// TwinCAT 3 PLC project ePU10V2
// ProgramVersion: 3.1.4026.24
// libraries:
//   Tc2_ControllerToolbox, * (Beckhoff Automation GmbH)
//   Tc2_EtherCAT, * (Beckhoff Automation GmbH)
//   Tc2_ModbusSrv, * (Beckhoff Automation GmbH)
//   Tc2_ProfinetDiag, * (Beckhoff Automation GmbH)
//   Tc2_Standard, * (Beckhoff Automation GmbH)
//   Tc2_SUPS, * (Beckhoff Automation GmbH)
//   Tc2_System, * (Beckhoff Automation GmbH)
//   Tc2_Utilities, * (Beckhoff Automation GmbH)
//   Tc3_EventLogger, * (Beckhoff Automation GmbH)
//   Tc3_IotBase, * (Beckhoff Automation GmbH)
//   Tc3_JsonXml, * (Beckhoff Automation GmbH)
// project tree:
//   DUTs/Enums/ eBatteryType.TcDUT, eForceBool.TcDUT, eGridTripMode.TcDUT, eObject_ID.TcDUT, ePNcouplerType.TcDUT, eSubValues.TcDUT, Phases.TcDUT
//   DUTs/Structs/ ST_AnalogInputData.TcDUT, ST_AnalogInputDiag.TcDUT, ST_Service_DigitalOutIn.TcDUT, ST_Service_DigitalOutInWithDependency.TcDUT, ST_Service_DigitalOutInWithSafety.TcDUT
//   DUTs/System/ ST_System_Config.TcDUT, ST_System_GridcodeParams.TcDUT, ST_System_MachineParams.TcDUT
//   GVLs/ Service.TcGVL, GVL.TcGVL, Settings.TcGVL, Units.TcGVL
//   POUs/Eventlogger/_enum/ eEventLogCategory.TcDUT, eEventLogSeverity.TcDUT
//   POUs/Eventlogger/_structs/ ST_EventLogEntry.TcDUT, ST_EventLogger_Params.TcDUT
//   / PlcTask.TcTTO, MonitorControlTask.TcTTO
//   POUs/ErrorHandling/ ErrorHandling.TcPOU, FB_AddErrorST.TcPOU
//   POUs/ErrorHandling/_enums/ eErrAckAccess.TcDUT, eSeverity.TcDUT
//   POUs/ErrorHandling/_strucs/ ST_ErrorStruct.TcDUT
//   POUs/Functions-FBs-Programs/ fbValueOutOfRange.TcPOU, Fb_BindControlVars.TcPOU, fb_IncrementPowerStep.TcPOU, FB_OverCurrentDetect.TcPOU, fb_Ramp.TcPOU, fb_Ramp_dual.TcPOU, FB_UpperLimitAndTimeExceeded.TcPOU, ITF_StandardFB.TcIO
//   POUs/Functions-FBs-Programs/IO_modules/Beckhoff/ FB_EK1100.TcPOU, FB_EL3453.TcPOU
//   POUs/Functions-FBs-Programs/IO_modules/Beckhoff/Structs/ DataSelector.TcDUT, ST_PQGridQualityData.TcDUT, ST_PQPowerData.TcDUT, ST_PQstatusData.TcDUT, ST_PQVoltageData.TcDUT
//   POUs/Functions-FBs-Programs/_acFunctions/ AcCheck.TcPOU, ACFrequencyCheck.TcPOU, AcPhasesOK.TcPOU, ACVoltageCheck.TcPOU, CurrentToKw.TcPOU, fb_LOMdetection.TcPOU, kWToCurrent.TcPOU, LineUnbalance.TcPOU, PowerFactor.TcPOU, ReactivePower.TcPOU
//   POUs/Functions-FBs-Programs/_generalFunctions/ Between.TcPOU, ConcatMultiString.TcPOU, fb_MovingAverage.TcPOU, FB_StartStop.TcPOU, F_RoundReal.TcPOU, IsNaN.TcPOU, LimitTrigger.TcPOU, Median.TcPOU, PackByte.TcPOU, PackWord.TcPOU, Scale.TcPOU, ValueOutOfRange.TcPOU, WriteOnEdge.TcPOU, XNOR.TcPOU
//   POUs/Functions-FBs-Programs/_PRGS/ SystemClock.TcPOU
//   POUs/ MAIN_Fast.TcPOU, MAIN_Slow.TcPOU
//   POUs/MonitoringControl/ ControlManager.TcPOU, FB_TestScripts.TcPOU
//   POUs/MonitoringControl/ExternalControl/enums/ eExternalControlMode.TcDUT, GenGridMode.TcDUT, uSWversion.TcDUT
//   POUs/MonitoringControl/ExternalControl/ FB_ExtControllerTest.TcPOU, FB_ExternalController.TcPOU
//   POUs/MonitoringControl/ExternalControl/Structs/future use/ ST_PNInput_DCBusExpansion.TcDUT, ST_PNInput_DCCharger.TcDUT, ST_PNInput_ParallelOperation.TcDUT, ST_PNOutput_DCCharger.TcDUT, ST_PNOutput_DCExpansion.TcDUT, ST_PNOutput_ParallelOperation.TcDUT
//   POUs/MonitoringControl/ExternalControl/Structs/NestedStructs/ ST_PNInput_ACDCCharger.TcDUT, ST_PNInput_Battery.TcDUT, ST_PNInput_GenControl.TcDUT, ST_PNInput_General.TcDUT, ST_PNInput_InputField.TcDUT, ST_PNInput_InputGridControl.TcDUT, ST_PNInput_PeakShaveBox.TcDUT, ST_PNInput_Powerstack.TcDUT, ST_PNOutput_ACDCCharger.TcDUT, ST_PNOutput_Battery.TcDUT, ST_PNOutput_GenControl.TcDUT, ST_PNOutput_General.TcDUT, ST_PNOutput_InputField.TcDUT, ST_PNOutput_InputGridControl.TcDUT, ST_PNOutput_OutputField.TcDUT, ST_PNOutput_PeakShaveBox.TcDUT, ST_PNOutput_PowerStack.TcDUT, ST_PNOutput_ZPT.TcDUT
//   POUs/MonitoringControl/ExternalControl/Structs/ ST_Extcontroller_params.TcDUT, ST_PNinput.TcDUT, ST_PNOutput.TcDUT, ST_PNTest.TcDUT
//   POUs/MonitoringControl/HMI/ FB_HMIButtons.TcPOU, HMI.TcPOU
//   POUs/MonitoringControl/HMI/_Structs/ControlStructures/HardSettings %28localOnly%29/ ST_HardSettings.TcDUT (not stored), ST_HardSettings_DCcharger.TcDUT (not stored), ST_HardSettings_ParallelOperation.TcDUT (not stored), ST_HardSettings_PeakshaveBox.TcDUT (not stored), ST_HardSettings_Setup.TcDUT (not stored), ST_HardSettings_System.TcDUT (not stored)
//   POUs/MonitoringControl/HMI/_Structs/ControlStructures/OperationVars/ ST_OperationVars.TcDUT, ST_OperationVars_BMS.TcDUT, ST_OperationVars_DCcharger.TcDUT, ST_OperationVars_Genset.TcDUT, ST_OperationVars_Grid.TcDUT, ST_OperationVars_ParallelOperation.TcDUT, ST_OperationVars_System.TcDUT
//   POUs/MonitoringControl/HMI/_Structs/ControlStructures/SoftSettings %28Local+Extern%29/NestedStructs/ ST_Genset_params.TcDUT (not stored), ST_Genset_setpoints.TcDUT (not stored), ST_Input_breakersettings.TcDUT (not stored), ST_Loadbank_params.TcDUT (not stored), ST_peakshave_setpoints.TcDUT (not stored), ST_ScheduleTimeSlot.TcDUT (not stored)
//   POUs/MonitoringControl/HMI/_Structs/ControlStructures/SoftSettings %28Local+Extern%29/ ST_SoftSettings.TcDUT (not stored), ST_Softsettings_AcDcCharger.TcDUT (not stored), ST_SoftSettings_DcLink.TcDUT (not stored), ST_SoftSettings_Genset.TcDUT (not stored), ST_SoftSettings_Grid.TcDUT (not stored), ST_SoftSettings_PeakshaveBox.TcDUT (not stored), ST_SoftSettings_Setup.TcDUT (not stored), ST_SoftSettings_System.TcDUT (not stored)
//   POUs/MonitoringControl/HMI/_Structs/ControlStructures/ ST_ControlsHMIonly.TcDUT, ST_ControlVars.TcDUT
//   POUs/MonitoringControl/HMI/_Structs/MonitoringStructures/ ST_HMIdata.TcDUT, ST_HMI_ConditionalFormatting.TcDUT, ST_HMI_Monitor_AcDcCharger.TcDUT, ST_HMI_Monitor_Arraydata.TcDUT, ST_HMI_Monitor_ArrayDataFormat.TcDUT, ST_HMI_Monitor_Battery.TcDUT, ST_HMI_Monitor_Connections.TcDUT, ST_HMI_Monitor_CoolingSystem.TcDUT, ST_HMI_Monitor_DcLink.TcDUT, ST_HMI_Monitor_Enclosure.TcDUT, ST_HMI_Monitor_FireDetection.TcDUT, ST_HMI_Monitor_IPSU.TcDUT, ST_HMI_Monitor_Limits.TcDUT, ST_HMI_Monitor_OCP.TcDUT, ST_HMI_Monitor_Powerstack.TcDUT, ST_HMI_Monitor_Protections.TcDUT, ST_HMI_Monitor_PSB.TcDUT, ST_HMI_Monitor_switchgear.TcDUT, ST_HMI_Monitor_System.TcDUT, ST_HMI_Monitor_UPS.TcDUT, ST_HMI_Monitor_ZPT.TcDUT, ST_HMI_PowerMeas.TcDUT, ST_HMI_PowerMeasDC.TcDUT
//   POUs/MonitoringControl/HMI/_Structs/ ST_HMI_Control.TcDUT, ST_HMI_Historize.TcDUT, ST_HMI_Monitor.TcDUT
//   POUs/MonitoringControl/IoT/DUTS/ eConnectionState.TcDUT, eDataMappingVarNames.TcDUT, eIoTCommVersion.TcDUT, eLogType.TcDUT, eUpdate.TcDUT, e_ORAttributeType.TcDUT, ST_AutoProvisioning.TcDUT, ST_IotProps.TcDUT, ST_RW.TcDUT, ST_Supervisor.TcDUT, ST_VarBuffer.TcDUT
//   POUs/MonitoringControl/IoT/ FB_IotController.TcPOU, MqttComOpenremote.TcPOU, RestComOpenremote.TcPOU
//   POUs/MonitoringControl/IoT/_Structs/ ST_IoTDataHMI.TcDUT, ST_IotData_credits.TcDUT, st_IOT_params.TcDUT, ST_IOT_SentStateLog.TcDUT
//   POUs/MonitoringControl/_Enums/ eAcInputType.TcDUT, eCapTestSTate.TcDUT, eControlSources.TcDUT, eDcInputType.TcDUT, eEarthingSystems.TcDUT, eGridFormingMode.TcDUT, eGridMode.TcDUT, eNetContactorDirection.TcDUT, eOperationMode.TcDUT, ePeakshaveMode.TcDUT, ePowerControlType.TcDUT, eSchedulerMode.TcDUT, eSystemState.TcDUT, eUgridPowerMode.TcDUT
//   POUs/MonitoringControl/_Structs/ ST_ExtController_Events.TcDUT, ST_ExtController_get.TcDUT, ST_ExtController_limits.TcDUT, ST_ExtController_Set.TcDUT, ST_PLCPersistentVars.TcDUT
//   POUs/Objects/4Grouter/Struct/ ST_router_service.TcDUT, dwtoreal.TcDUT, eModemState.TcDUT, eNetworkState.TcDUT, eSimSelectionMode.TcDUT, eSimState.TcDUT, eSMSStatus.TcDUT, eWifiSecurityTypes.TcDUT, eWifiStatus.TcDUT, st_Device.TcDUT, st_GPS.TcDUT, st_mobile.TcDUT, st_Router_Events.TcDUT, st_router_get.TcDUT, ST_Router_params.TcDUT, ST_Router_set.TcDUT, st_Wifi.TcDUT
//   POUs/Objects/ACDCCharger/Structs/ ST_ACDCCharger_Service.TcDUT, ST_ACDCCharger_events.TcDUT, ST_ACDCCharger_get.TcDUT, ST_ACDCCharger_params.TcDUT, ST_ACDCCharger_set.TcDUT, ST_SystemDiagnostic.TcDUT, ST_SystemEval.TcDUT
//   POUs/Objects/BMS/eNums/ eBMS_Status.TcDUT, eHVDC_Powerstatus.TcDUT, ePOUState.TcDUT, ePowerControl.TcDUT, ePowerOnStatus.TcDUT
//   POUs/Objects/BMS/ FB_BMS.TcPOU, FB_BMS_IO.TcPOU
//   POUs/Objects/BMS/Structs/ st_BMS_BatterySummary.TcDUT, st_BMS_Events.TcDUT, st_BMS_Get.TcDUT, st_BMS_Params.TcDUT, ST_BMS_Service.TcDUT, st_BMS_Set.TcDUT, st_MBMU_BatterySummary.TcDUT, st_MBMU_Status.TcDUT, st_SBMU_BatterySummary.TcDUT, st_SBMU_Status.TcDUT
//   POUs/Objects/CoolingSystem/enums/ eConditioningRequirement.TcDUT, eCoolingSystemState.TcDUT, eHeatPumpMode.TcDUT, eHeatPumpState.TcDUT, eSupportedHeatpumps.TcDUT
//   POUs/Objects/CoolingSystem/ FB_CoolingSystem.TcPOU, FB_LGThermaV.TcPOU, ITF_Heatpump.TcIO
//   POUs/Objects/CoolingSystem/structs/ LG_Coils.TcDUT, LG_ControlRegs.TcDUT, LG_InputRegs.TcDUT, LG_Statusbits.TcDUT, ST_CoolingSystem_Events.TcDUT, ST_CoolingSystem_Get.TcDUT, ST_CoolingSystem_MaintenanceParams.TcDUT, ST_Coolingsystem_params.TcDUT, ST_HeatpumpData.TcDUT, ST_HeatPumpEvents.TcDUT, ST_HeatPump_Get.TcDUT, st_TCME31_get_1.TcDUT, st_TCME31_Set_1.TcDUT
//   POUs/Objects/DCLink/ FB_CNV520.TcPOU, FB_DCLink.TcPOU, FB_ShuntBournsSSD.TcPOU
//   POUs/Objects/DCLink/_Enums/ eDcLinkState.TcDUT, eDCpowerPriority.TcDUT
//   POUs/Objects/DCLink/_Structs/ ST_Bourns_errors.TcDUT, ST_Bourns_Powerdata.TcDUT, ST_DCLink_events.TcDUT, ST_DCLink_Get.TcDUT, ST_DCLink_IO.TcDUT, ST_DCLink_params.TcDUT, ST_DCLink_set.TcDUT, st_Pixsys.TcDUT
//   POUs/Objects/PowerQualityMonitor/ FB_EastronSDM630.TcPOU, FB_PowerQualityMonitoring.TcPOU
//   POUs/Objects/PowerQualityMonitor/_Enums/ eACRotationState.TcDUT
//   POUs/Objects/PowerQualityMonitor/_Structs/ ST_PowerMonitor_BESS.TcDUT, ST_PowerMonitor_Events.TcDUT, ST_PowerMonitor_get.TcDUT, ST_PowerMonitor_InputField.TcDUT, ST_PowerMonitor_OutputField.TcDUT
//   POUs/Objects/PowerStack/NetContactor/_Structs/ ST_Netcontactor_service.TcDUT, ST_Netcontactor_Events.TcDUT, ST_Netcontactor_get.TcDUT, ST_Netcontactor_set.TcDUT
//   POUs/Objects/PowerStack/_Structs/ ST_Powermodule_Service.TcDUT, ST_Powerstack_MaintenanceParams.TcDUT, ST_Powerstack_Service.TcDUT, ST_PowerModule_calibration.TcDUT, ST_PowerModule_get.TcDUT, ST_PowerModule_params.TcDUT, ST_PowerModule_set.TcDUT, ST_Powerstack_Calibration.TcDUT, ST_PowerStack_get.TcDUT, ST_Powerstack_LOMParams.TcDUT, ST_PowerStack_params.TcDUT, ST_PowerStack_Set.TcDUT
//   POUs/Safety/ Safety.TcPOU, ST_Safety_ContactorEDM.TcDUT, ST_Safety_get.TcDUT, ST_Safety_ToSafetyPrg.TcDUT
//   POUs/Objects/4Grouter/ FB_Teltonika.TcPOU
//   POUs/Objects/ACDCCharger/Enums/ eAcDcChargerState.TcDUT
//   POUs/Objects/ACDCCharger/ FB_AcDcCharger.TcPOU
//   POUs/Objects/ACDCCharger/Structs/Hadi/ E_ChargerState.TcDUT, ST_CanId.TcDUT, ST_ChargerControl.TcDUT, ST_Control.TcDUT, ST_Data.TcDUT, ST_ModuleControl.TcDUT, ST_ModuleData.TcDUT, ST_ModuleStatus.TcDUT
//   POUs/Objects/ACSwitchgear %28clientbox%29/ FB_ACSwitchgear.TcPOU (not stored), ST_ACswitchgear_events.TcDUT (not stored), ST_ACSwitchgear_Get.TcDUT (not stored), ST_ACswitchgear_IO.TcDUT (not stored), ST_ACswitchgear_params.TcDUT (not stored), ST_ACswitchgear_set.TcDUT (not stored)
//   POUs/Objects/Enclosure/Climate/ FB_EnclosureClimate.TcPOU, ST_Enclosureclimate_events.TcDUT, ST_EnclosureClimate_get.TcDUT, ST_EnclosureClimate_Params.TcDUT
//   POUs/Objects/Enclosure/Doors/ FB_DoorsNLocks.TcPOU, ST_DoorsNLocks_get.TcDUT
//   POUs/Objects/Enclosure/ FB_Enclosure.TcPOU
//   POUs/Objects/Enclosure/LedIndicator/BeckhoffController/ eDCstate.TcDUT, eLEDSteps.TcDUT, eSystemStatus.TcDUT, FB_LedBeckhoff.TcPOU, LEDColor.TcDUT, LEDCommands.TcDUT, LEDControl.TcDUT, LEDStatus.TcDUT
//   POUs/Objects/Enclosure/LedIndicator/ eColorOrder.TcDUT, FB_Ledstrip.TcPOU, ST_Ledstrip_get.TcDUT, st_Ledstrip_MachineData.TcDUT, st_Ledstrip_params.TcDUT
//   POUs/Objects/Enclosure/_struct/ ST_Enclosure_get.TcDUT, st_Enclosure_params.TcDUT, ST_enclosure_set.TcDUT
//   POUs/Objects/GenComm/eNums/ eGenControlProtocol.TcDUT, eGenOperationMode.TcDUT, eOnOffState.TcDUT
//   POUs/Objects/GenComm/ FB_AGC150.TcPOU, FB_GenComm.TcPOU
//   POUs/Objects/GenComm/Structs/ ST_AGC150_Set.TcDUT, ST_GenComm_Params.TcDUT, ST_Genset_Get.TcDUT, ST_Genset_Set.TcDUT
//   POUs/Objects/HartingIO/ FB_HartingIO.TcPOU, ST_HartingIO_get.TcDUT, ST_HartingIO_params.TcDUT, ST_HartingIO_set.TcDUT
//   POUs/Objects/HartingIO/_Enum/ eAOTarget.TcDUT, eInputSignal.TcDUT, eOutputContactSignal.TcDUT
//   POUs/Objects/InterMachineCom/ FB_ConnectMqttBroker.TcPOU, FB_InterMachineCommunication.TcPOU, ST_InterMachineCom_Master.TcDUT, ST_IntermachineCom_params.TcDUT, st_InterMachineCom_Slave.TcDUT, ST_InterMachineCom_SlaveConData.TcDUT
//   POUs/Objects/InternalPowerSupply/eNums/ e400VSupplySource.TcDUT, eSupplyState.TcDUT
//   POUs/Objects/InternalPowerSupply/ FB_InternalPowerSupply.TcPOU, FB_InternalPowerSupply_IO.TcPOU
//   POUs/Objects/InternalPowerSupply/Structs/ ST_InternalPowerStatus.TcDUT, ST_InternalPowerSupply_Events.TcDUT, ST_InternalPowerSupply_Get.TcDUT, ST_InternalPowerSupply_Params.TcDUT, ST_InternalPowerSupply_PowerDemand.TcDUT
//   POUs/Objects/InternalPowerSupply/UPS/eNums/ eUPSState.TcDUT
//   POUs/Objects/InternalPowerSupply/UPS/ FB_UPS.TcPOU
//   POUs/Objects/InternalPowerSupply/UPS/Structs/ ST_UPSData.TcDUT, ST_UPSEvents.TcDUT, ST_UPSGET.TcDUT
//   POUs/Objects/NeutralTransformer/ FB_NeutralTransformer.TcPOU, FB_NeutralTransformer_IO.TcPOU
//   POUs/Objects/NeutralTransformer/_Struct/ ST_NeutralTransformer_events.TcDUT, ST_NeutralTransformer_Get.TcDUT, ST_Neutraltransformer_params.TcDUT
//   POUs/Objects/PeakshaveBox/DUTs/ ePSBMode.TcDUT
//   POUs/Objects/PeakshaveBox/ FB_PeakshaveBox.TcPOU, ST_PeakShaveBox_Get.TcDUT, ST_peakshavebox_params.TcDUT, ST_PeakshaveBox_Set.TcDUT
//   POUs/Objects/PLCStatus/Enum/ eFTPState.TcDUT, eInstalState.TcDUT, eNetcomState.TcDUT
//   POUs/Objects/PLCStatus/ FB_PLCState.TcPOU, FB_PLCUpdate.TcPOU, ST_EL9410.TcDUT, ST_PLCstate_get.TcDUT, ST_PLC_events.TcDUT
//   POUs/Objects/PowerStack/ FB_PowerStack.TcPOU
//   POUs/Objects/PowerStack/NetContactor/ eNetcontMode.TcDUT, FB_NetContactor.TcPOU, FB_NetContactor_IO.TcPOU
//   POUs/Objects/PowerStack/PowerModule/ FB_PowerModule.TcPOU, FB_Powermodule_additionalMeasurements.TcPOU, FB_PowerModule_Buscoupler.TcPOU, FB_PowerModule_Inverter.TcPOU
//   POUs/Objects/PowerStack/_Enums/ eInverterModes.TcDUT, eNetContactorState.TcDUT, ePLM.TcDUT, ePowerModes.TcDUT, ePowerModuleThrottlingState.TcDUT, ePowerstate.TcDUT, eStatusPowerModule.TcDUT, eStatusPowerStack.TcDUT
//   POUs/Objects/PowerStack/_Structs/NestedStructs/ ST_InverterControlWord.TcDUT, ST_Inverter_additionalTemperatures.TcDUT, ST_Inverter_LineState.TcDUT, ST_Inverter_StatusWord.TcDUT, ST_Inverter_UgridStatusWord.TcDUT, ST_Inverter_Write.TcDUT, ST_Powermodule_CalibData.TcDUT, ST_Powermodule_Events.TcDUT, ST_Powermodule_PowerCurveCoefficients.TcDUT, ST_PowerStack_Events.TcDUT, ST_Powerstack_ShiftingParams.TcDUT
//   POUs/Objects/ProtectionSystems/ FB_ProtectionSystems.TcPOU
//   POUs/Objects/ProtectionSystems/FireDetection/ FB_FireDetection.TcPOU, FB_FireDetection_IO.TcPOU
//   POUs/Objects/ProtectionSystems/FireDetection/_Enums/ eCOAlarmStatus.TcDUT, eSmokeDetectAlarmStatus.TcDUT
//   POUs/Objects/ProtectionSystems/FireDetection/_Structs/ ST_CODetectors.TcDUT, ST_FireDetection_get.TcDUT, st_Firedetection_params.TcDUT, ST_FireDetection_set.TcDUT, ST_FireSystem_Events.TcDUT, ST_SmokeDetectors.TcDUT, ST_SmokeDetIO.TcDUT
//   POUs/Objects/ProtectionSystems/InsulationMonitoring/ FB_InsulationMonitor.TcPOU
//   POUs/Objects/ProtectionSystems/InsulationMonitoring/_Structs/ ST_InsulationMonitor_get.TcDUT, ST_InsulationMonitor_params.TcDUT, St_InsulationMonitor_PassThrough.TcDUT, ST_InsulationMonitor_set.TcDUT
//   POUs/Objects/ProtectionSystems/OvercurrentProtection/ FB_OvercurrentProtection.TcPOU
//   POUs/Objects/ProtectionSystems/OvercurrentProtection/_Structs/ ST_OvercurrentProtection_Events.TcDUT, ST_OvercurrentProtection_get.TcDUT, ST_OvercurrentProtection_InternalLinking.TcDUT, ST_OvercurrentProtection_Params.TcDUT, ST_OvercurrentProtection_set.TcDUT
//   POUs/Objects/ProtectionSystems/ResidualCurrentMonitoring/ FB_RCMonitor.TcPOU
//   POUs/Objects/ProtectionSystems/ResidualCurrentMonitoring/_Structs/ ST_ResidualCurrentMonitor_get.TcDUT
//   POUs/Objects/ProtectionSystems/SurgeProtection/ FB_SurgeProtection.TcPOU
//   POUs/Objects/ProtectionSystems/SurgeProtection/_Structs/ ST_Surgeprotection_get.TcDUT
//   POUs/Objects/ProtectionSystems/_Struct/ ST_ProtectionSystems_get.TcDUT, ST_ProtectionSystems_Params.TcDUT, ST_ProtectionSystems_set.TcDUT
//   POUs/Objects/RemoteIO/ FB_TruCompTCME21_IOModule.TcPOU, st_TCME31_get.TcDUT, st_TCME31_Set.TcDUT
//   POUs/Objects/WearLogging/ eEntryType.TcDUT, eLogItemGroupID.TcDUT, eLogTypes.TcDUT, FB_Varlogger.TcPOU, LogState.TcDUT, WearLogging.TcPOU
//   POUs/System/ FB_SystemControl.TcPOU
//   POUs/Eventlogger/ FB_Eventlogger.TcPOU, FB_EventLogClient.TcPOU
//   POUs/System/GenGridControl/ FB_ContactorControl.TcPOU, FB_GenGridController.TcPOU
//   POUs/System/GenGridControl/_enums/ eBreakerOperationMode.TcDUT, eGenGridState.TcDUT, eGenIsoInverterMode.TcDUT, eGensetMode.TcDUT, eGensetStartStop.TcDUT, ePowerControlMode.TcDUT, eRunCondition.TcDUT
//   POUs/System/GenGridControl/_structs/ ST_ContactorControl_params.TcDUT, ST_GenGridController_Events.TcDUT, ST_GenGridController_get.TcDUT, ST_GenGridController_Params.TcDUT, St_GenGridController_ParamsGenset.TcDUT, ST_GenGridController_SyncData.TcDUT
//   POUs/System/PowerControl/ fb_measurementCheck.TcPOU, FB_PowerControl.TcPOU
//   POUs/System/PowerControl/_enums/ ePIDmode.TcDUT
//   POUs/System/PowerControl/_Structs/ ST_PowerControl_Events.TcDUT, ST_PowerControl_Get.TcDUT, st_Powercontrol_params.TcDUT, st_Powercontrol_PIDparams.TcDUT, ST_PowerControl_PsTarget_Measurements.TcDUT, ST_Powercontrol_set.TcDUT, ST_PowerControl_SocDroopParams.TcDUT, ST_PowerControl_Target.TcDUT
//   POUs/System/_Structs/ ST_SystemTime.TcDUT, ST_System_Calibration.TcDUT, ST_System_Control.TcDUT, ST_System_Events.TcDUT, ST_System_get.TcDUT, ST_System_Monitor.TcDUT, ST_System_params.TcDUT, ST_System_Properties.TcDUT, ST_System_set.TcDUT
// real-time tasks:
//   TASK FastTask: cycle T#1ms, priority 4, ADS port 350
//   TASK SlowTask: cycle T#10ms, priority 8, ADS port 351
// I/O:
//   DEVICE InternalBus (EtherCAT), AmsNetId 10.46.35.98.2.1
//     Main PLC [EK1200-5000 EtherCAT Power supply (2A E-Bus)]
//       Term 34 (EL6070-0033) [EL6070-0033 1Ch. Licence key terminal, individual licences]
//       Term 2 (EL1809) [EL1809 16Ch. Dig. Input 24V, 3ms]
//       Term 3 (EL2809) [EL2809 16Ch. Dig. Output 24V, 0.5A]
//       Term 4 (EL2809) [EL2809 16Ch. Dig. Output 24V, 0.5A]
//       Term 38 (EL3124-0090) [EL3124-0090 4Ch. Ana. Input 4-20mA, Diff., TwinSAFE SC]
//         modules: Module 1 (TwinSAFE Single Channel)
//       Term 6 (EL3214) [EL3214 4Ch. Ana. Input PT100 (RTD)]
//       Term 7 (EL2574) [EL2574 4 Ch. Pixel LED Controller] (disabled)
//         modules: SlotGroup 1 (Slot 1, 2), SlotGroup 1 (Slot 1, 2), SlotGroup 1 (Slot 1, 2), SlotGroup 1 (Slot 1, 2), SlotGroup 2 (Slot 3, 4), SlotGroup 2 (Slot 3, 4), SlotGroup 2 (Slot 3, 4), SlotGroup 2 (Slot 3, 4)
//       Term 9 (EL1918) [EL1918, 8Ch. Safety Input 24V, TwinSAFE]
//         modules: Module 2 (FSLOGIC)
//       Term 10 (EL2904) [EL2904, 4 Ch. Safety Output 24V, 0.5A, TwinSAFE]
//         modules: Module 1 (FSOES), Module 2 (DO)
//       Term 11 (EK1122) [EK1122 2 port EtherCAT junction]
//       Term 12 (EL9011) [EL9011 End Terminal]
//     Clientpanel-input-IO [EK1101 EtherCAT Coupler (2A E-Bus, ID switch)]
//       Term 26 (EL3453-0020) [EL3453 3Ch. Power Measuring calibrated]
//       Term 27 (EL9011) [EL9011 End Terminal]
//     Doorswitch-IO [EK1101 EtherCAT Coupler (2A E-Bus, ID switch)]
//       Term 24 (EL1008) [EL1008 8Ch. Dig. Input 24V, 3ms]
//       Term 25 (EL9011) [EL9011 End Terminal]
//     Clientpanel-output-IO [EK1101 EtherCAT Coupler (2A E-Bus, ID switch)]
//       Term 13 (EL3453-0020) [EL3453 3Ch. Power Measuring calibrated]
//       Term 21 (EL1809) [EL1809 16Ch. Dig. Input 24V, 3ms]
//       Term 22 (EL2809) [EL2809 16Ch. Dig. Output 24V, 0.5A]
//       Term 23 (EL9011) [EL9011 End Terminal]
//     ACDCcharger-IO [EK1101 EtherCAT Coupler (2A E-Bus, ID switch)]
//       Term 28 (EL6751) [EL6751 CANopen Master]
//       Term 29 (EL9011) [EL9011 End Terminal]
//   DEVICE Device 2 (Profinet Controller), AmsNetId 10.46.35.98.3.1
//     quint4-ups [Phoenix Contact PROFINET IO - Uninterruptible Power Supply 2907079]
//       modules: Term 5 (DAP Module), Term 6 (QUINT4-UPS 24DC/40)
//     pm1buscoupler [Beckhoff Automation PROFINET I/O - EtherCAT coupler, IRT, V2.43, port diagnostic, shared device and system redundancy supported EK9320]
//       modules: Term 1 (DAP Module), Term 3 (EL1008), Term 2 (EL2008), Term 8 (EL3208), Term 8 (EL3208)_1, Term 8 (EL3208)_2, Term 8 (EL3208)_3, Term 8 (EL3208)_4
//     arfif106-1 [VACON VACON OPTE9 Dual-port Ethernet OPTE9]
//       modules: Term 7 (DAP Module), Term 4 (Vendor 4 + 16 PD)
//   DEVICE Device 3 (EL6751), AmsNetId 10.46.35.98.4.1
//     Box 1 (CAN Interface)
//   DEVICE ExternalBus (EtherCAT), AmsNetId 10.46.35.98.5.1
//     PSB_V1 [EK1101 EtherCAT Coupler (2A E-Bus, ID switch)]
//       Term 31 (EL3453) [EL3453 3Ch. Power Measuring]
//       Term 32 (EL9011) [EL9011 End Terminal]
// variable links:
//   InternalBus (EtherCAT) <-> InternalBus (EtherCAT)/Main PLC/Term 10 (EL2904)
//     Main PLC/Term 9 (EL1918)/ConnectionInputs/TwinSafeGroup1.Term 10 (EL2904) - Module 1 (FSOES)_13 TxPDO <-> Module 1 (FSOES)/RxPDO/FSOE
//     Main PLC/Term 9 (EL1918)/ConnectionOutputs/TwinSafeGroup1.Term 10 (EL2904) - Module 1 (FSOES)_13 RxPDO <-> Module 1 (FSOES)/TxPDO/FSOE
//   InternalBus (EtherCAT) <-> InternalBus (EtherCAT)/Main PLC/Term 9 (EL1918)
//     Main PLC/Term 38 (EL3124-0090)/Module 1 (TwinSAFE Single Channel)/TSC Inputs/TSC <-> ConnectionOutputs/TwinSafeGroup1.Term 38 (EL3124-0090) - Module 1 (TwinSAFE Single Channel)_15 RxPDO
//     Main PLC/Term 38 (EL3124-0090)/Module 1 (TwinSAFE Single Channel)/TSC Outputs/TSC <-> ConnectionInputs/TwinSafeGroup1.Term 38 (EL3124-0090) - Module 1 (TwinSAFE Single Channel)_15 TxPDO

CONFIGURATION ePU10V2
    RESOURCE PLC ON TwinCAT3
        TASK PlcTask(INTERVAL := T#1ms, PRIORITY := 4);
        TASK MonitorControlTask(INTERVAL := T#10ms, PRIORITY := 8);
        PROGRAM MAIN_Fast WITH PlcTask : MAIN_Fast;
        PROGRAM MAIN_Slow WITH MonitorControlTask : MAIN_Slow;
    END_RESOURCE
END_CONFIGURATION

// ---- DUTs/Enums/eBatteryType.TcDUT
{attribute 'qualified_only'}
{attribute 'strict'}
TYPE eBatteryType :
(
	standard_306Ah := 0,
	highpower_280Ah := 1
);
END_TYPE

// ---- DUTs/Enums/eForceBool.TcDUT
{attribute 'qualified_only'}
{attribute 'strict'}
{attribute 'to_string'}
TYPE eForceBool:
(
	none := 0,
	On	:= 1,
	Off := 2
);
END_TYPE

// ---- DUTs/Enums/eGridTripMode.TcDUT
{attribute 'qualified_only'}
{attribute 'strict'}
TYPE eGridTripMode :
(
	Gridcode := 500,
	Default	:= 30,
	UPS		:= 10	
) UINT; //milliseconds
END_TYPE

// ---- DUTs/Enums/eObject_ID.TcDUT
{attribute 'qualified_only'}
{attribute 'to_string'}
TYPE eObject_ID :
(	
	None					:= 0,
	Safety					:= 10,
	PowerStack				:= 100,
	NetContactor			:= 150,
	PowerModuleMaster 		:= 200,
	PowerModuleSlave 		:= 300,
	PowerMonitor			:= 400,
	InternalPowerSupply		:= 500,
	UPS						:= 550,
	NeutralTransformer		:= 600,
	HartingIO				:= 650,
	Battery					:= 700,
	Cooling					:= 800,
	HeatPump				:= 850,
	AC_Switchgear			:= 900,
	DC_Switchgear			:= 950,
	RCM						:= 1000,
	SurgeProtection			:= 1010,
	InsulationMonitor		:= 1020,
	Firedetection			:= 1030,
	OCP						:= 1050,
	Enclosure_LED			:= 1200,
	Enclosure_doors			:= 1210,
	Enclosure_climate		:= 1220,
	PLC						:= 2000,
	Router					:= 2100,
	PNcontroller			:= 2200,
	IotController			:= 2300,
	PeakshaveBox			:= 2400,
	ACDCCharger				:= 2500,
	RemoteIO				:= 2600,
	GenGridController		:= 3000,
	PowerController			:= 3100,
	System					:= 3200,
	Genset					:= 4000
	
) WORD := None;
END_TYPE

// ---- DUTs/Enums/ePNcouplerType.TcDUT
{attribute 'qualified_only'}
{attribute 'strict'}

TYPE ePNcouplerType :
(
	None := 0,
	ModbusTCP:= 1,
	Profinet := 2,
	ModbusTCPV2 := 3
);
END_TYPE

// ---- DUTs/Enums/eSubValues.TcDUT
{attribute 'qualified_only'}
{attribute 'strict'}
TYPE eSubValues :
(
	Minimum := 0,
	Average := 1,
	Maximum := 2
);
END_TYPE

// ---- DUTs/Enums/Phases.TcDUT
{attribute 'qualified_only'}
{attribute 'strict'}
{attribute 'to_string'}
TYPE Phases :
(
	AVG 		:= 0,
	L1 			:= 1,
	L2 			:= 2,
	L3 			:= 3,
	N 			:= 4,
	minimum		:= 5,
	maximum		:= 6,
	Sum			:= 7
) INT;
END_TYPE

// ---- DUTs/Structs/ST_AnalogInputData.TcDUT
TYPE ST_AnalogInputData :
STRUCT
	Value			: INT;
	Status			: ST_AnalogInputDiag;
END_STRUCT
END_TYPE

// ---- DUTs/Structs/ST_AnalogInputDiag.TcDUT
TYPE ST_AnalogInputDiag :
STRUCT
	Underrange			: BIT;
	Overrange			: BIT;
	Error				: BIT;
END_STRUCT 
END_TYPE

// ---- DUTs/Structs/ST_Service_DigitalOutIn.TcDUT
TYPE ST_Service_DigitalOutIn :
STRUCT
	Force				: eForceBool; //write value
	Feedback			: BOOL; // readvalue
END_STRUCT
END_TYPE

// ---- DUTs/Structs/ST_Service_DigitalOutInWithDependency.TcDUT
TYPE ST_Service_DigitalOutInWithDependency EXTENDS ST_Service_DigitalOutIn:
STRUCT
	{attribute 'TcHmiSystemEng.Parameter.Name' := 'Dependency state'}
	DependencyOK			: BOOL; 
END_STRUCT
END_TYPE

// ---- DUTs/Structs/ST_Service_DigitalOutInWithSafety.TcDUT
TYPE ST_Service_DigitalOutInWithSafety EXTENDS ST_Service_DigitalOutIn:
STRUCT
	{attribute 'TcHmiSystemEng.Parameter.Name' := 'Dependency state'}
	SafetyLoopOK			: BOOL; 
	EDM					: BOOL;
END_STRUCT
END_TYPE

// ---- DUTs/System/ST_System_Config.TcDUT
TYPE ST_System_Config :
STRUCT
	DefaultSettingsActive			: BOOL := TRUE; //To verify when all settings have been reset.
	b_DoublePowerModule				: BOOL := FALSE;
	b_PeakshaverBoxEnable			: BOOL := FALSE;
	
	//NeutralTransformer
	b_NeutralTransformer			: BOOL := FALSE;
	
	
	//Netcontactor
	b_AutomaticACrotation			: BOOL := FALSE;
	
	//DC
	b_DCbuscoupling					: BOOL := FALSE;
	b_DcCharger						: BOOL := FALSE;
	
	//AC
	b_ACInputConnection				: BOOL := FALSE;
	b_ThirdOutputConnection			: BOOL := FALSE;
	//communication
	e_PNcouplerType					: ePNcouplerType := ePNcouplerType.None;
	
	//batteries
	by_NoBatteryStrings			 	: BYTE := 3; // pieces
	e_BatteryType					: eBatteryType := eBatteryType.standard_306Ah;
	
	//Powernet option
	b_PowernetClient				: BOOL :=  FALSE;
	
	//CLIENT specifics
	b_ClientHMI						: BOOL := FALSE;
	
END_STRUCT
END_TYPE

// ---- DUTs/System/ST_System_GridcodeParams.TcDUT
TYPE ST_System_GridcodeParams :
STRUCT
	r_GridNominalVoltage				: REAL := 400; //VAC
	r_GridNominalFrequency				: REAL := 50; // Hz
	r_GridVoltageMin					: REAL := 360;
	r_GridvoltageMax					: REAL := 440;
	r_GridFrequencyMin					: REAL := 48.5;
	r_GridFrequencyMax					: REAL := 51.5;
	r_CurrentUnbalanceLimit				: REAL := 50;  //%
	ui_GCokReleaseTime					: UINT := 60; //seconds
	ui_GCTripMaxTripTime				: UINT := 40; // milliseconds
END_STRUCT
END_TYPE

// ---- DUTs/System/ST_System_MachineParams.TcDUT
TYPE ST_System_MachineParams :
STRUCT
	BMS									: ST_BMS_params;
	ACDCCharger							: ST_ACDCCharger_params;
	Interpowersupply					: ST_InternalPowerSupply_Params;
	Powerstack							: ST_Powerstack_Params;
	Coolingsystem						: ST_Coolingsystem_Params;
	NeutralTransformer					: ST_Neutraltransformer_Params;
	Protections							: ST_Protectionsystems_Params;
	Enclosure							: ST_Enclosure_Params;
	system								: ST_System_params;
	IOT									: ST_IOT_params;
	Router								: ST_Router_params;
	PSB									: ST_peakshavebox_params;
	ACswitchgear						: ST_ACswitchgear_params;
	HartingIO							: ST_HartingIO_params;
	GenComm								: ST_GenComm_params;
	Eventlogger							: ST_EventLogger_params;
	DC									: ST_DClink_params;
	ExtController						: ST_ExtController_params;
END_STRUCT
END_TYPE

// ---- POUs/Eventlogger/_enum/eEventLogCategory.TcDUT
{attribute 'qualified_only'}
{attribute 'strict'}
TYPE eEventLogCategory :
(
	Generic := 0,
	ReleaseTrigger := 1,
	SFCstep := 2,
	OperationMode := 3
);
END_TYPE

// ---- POUs/Eventlogger/_enum/eEventLogSeverity.TcDUT
{attribute 'qualified_only'}
{attribute 'strict'}
TYPE eEventLogSeverity :
(
	Info := 0,
	Warning := 1,
	Fault := 2
);
END_TYPE

// ---- POUs/Eventlogger/_structs/ST_EventLogEntry.TcDUT
TYPE ST_EventLogEntry :
STRUCT
	sTimestamp	: STRING(63);
	eCategory	: eEventLogCategory;
	eSeverity	: eEventLogSeverity;
	sSourceFB	: STRING(63);
	sMessage	: STRING(255);
END_STRUCT
END_TYPE

// ---- POUs/ErrorHandling/_enums/eErrAckAccess.TcDUT
{attribute 'qualified_only'}
{attribute 'strict'}
TYPE eErrAckAccess :
(
	General := 0,
	Operator := 1,
	VDL := 2
);
END_TYPE

// ---- POUs/ErrorHandling/_enums/eSeverity.TcDUT
{attribute 'qualified_only'}
{attribute 'to_string'}
TYPE eSeverity :
(
	None						:= 0,
	Info						:= 1,
	Warning 					:= 2,
	NormalShutdown				:= 3,
	QuickShutdown				:= 4,
	EmergencyShutdown			:= 5 //ONLY CALL FROM SAFETY PROGRAM		
);
END_TYPE

// ---- POUs/ErrorHandling/_strucs/ST_ErrorStruct.TcDUT
TYPE ST_ErrorStruct :
STRUCT
	b_ErrorActive	:BOOL;
	s_Severity 		:STRING(20);
	w_ID			:WORD;
	s_Message		:STRING(100);
	s_DateError		:STRING(20);
	s_TimeError		:STRING(20);
	s_TimeCleared	:STRING(20);
	b_SMSEnable		:BOOL;
END_STRUCT
END_TYPE

// ---- POUs/Eventlogger/_structs/ST_EventLogger_Params.TcDUT
TYPE  ST_EventLogger_Params :
STRUCT
	MaxFileSize 		: UDINT := 5000000; //bytes
	LogWriteInterval 	: TIME := T#1M;
	MaxFileCount 		: UINT := 100; 
	MaxFillGrade		: REAL := 0.9;  //controls how full a log file is allowed to get (as a percentage of MaxFileSize) before the logger rotates to the next file.
END_STRUCT
END_TYPE

// ---- POUs/Functions-FBs-Programs/IO_modules/Beckhoff/Structs/DataSelector.TcDUT
{attribute 'qualified_only'}
{attribute 'strict'}
TYPE DataSelector :
(
	_C 		:= 0,
	_V 		:= 1,
	_P		:= 2,
	_Q		:= 3,
	_S		:= 4,
	_E		:= 5,
	_F		:= 6	
);
END_TYPE

// ---- POUs/Functions-FBs-Programs/IO_modules/Beckhoff/Structs/ST_PQGridQualityData.TcDUT
TYPE ST_PQGridQualityData :
STRUCT
	b_systemState				: 	BOOL;
	uli_TimeVoltZeroCrossup 	: 	ULINT;
	r_PowerQualityFactor		:	REAL;
	r_ROCOF						: 	REAL;
END_STRUCT
END_TYPE

// ---- POUs/Functions-FBs-Programs/IO_modules/Beckhoff/Structs/ST_PQPowerData.TcDUT
TYPE ST_PQPowerData :
STRUCT
	//Power
	ar_ApparentPower			: 	ARRAY[0..3] OF REAL;
	ar_ReactivePower			: 	ARRAY[0..3] OF REAL;
	ar_ActivePower				: 	ARRAY[0..3] OF REAL;

	//Energy Consumed
	r_EnergyConsumed			:	REAL := 0;
	
	//Energy Delivered
	r_EnergySupplied			:	REAL := 0;
	
	//THD
	ar_CurrentTHD						:	ARRAY[0..3] OF REAL := [0, 0, 0, 0];	
	
	//PF
	ar_PowerFactor				:	ARRAY[0..3] OF REAL := [0, 0, 0, 0];
	
	//Current
	ar_Current					: 	ARRAY[0..4] OF REAL := [0, 0, 0, 0];
	r_CurrentUnbalance			:	REAL;
END_STRUCT
END_TYPE

// ---- POUs/Functions-FBs-Programs/IO_modules/Beckhoff/Structs/ST_PQstatusData.TcDUT
TYPE ST_PQstatusData:
STRUCT
	b_Fault			: BOOL;
	b_OverVoltage 	: BOOL;
	b_UnderVoltage	: BOOL;
	b_OverFrequency : BOOL;
	b_UnderFrequency: BOOL;
	b_OverCurrent	: BOOL;
	b_SettingFault	: BOOL;
	b_Error_Phase 	: ARRAY [1..3] OF BOOL;
END_STRUCT
END_TYPE

// ---- POUs/Functions-FBs-Programs/IO_modules/Beckhoff/Structs/ST_PQVoltageData.TcDUT
TYPE ST_PQVoltageData EXTENDS ST_PQPowerData:
STRUCT
	b_VoltagesOK			: 	BOOL;
	e_ACrotationStatus		:	eACRotationState;
	ar_PhaseVoltage			: 	ARRAY[0..3] OF REAL;
	ar_LineVoltage			:	ARRAY[0..3] OF REAL;
	ar_Frequency			: 	ARRAY[0..3] OF REAL;
	r_VoltageUnbalance		: 	REAL;
	ar_VoltageTHD			: 	ARRAY[0..3] OF REAL;
END_STRUCT
END_TYPE

// ---- POUs/MonitoringControl/ExternalControl/enums/eExternalControlMode.TcDUT
{attribute 'qualified_only'}
{attribute 'strict'}
TYPE eExternalControlMode :
(
	off := 0,
	Readonly := 1,
	BasicControl := 2,
	AdvancedControl := 3
);
END_TYPE

// ---- POUs/MonitoringControl/ExternalControl/enums/GenGridMode.TcDUT
{attribute 'qualified_only'}
{attribute 'strict'}
TYPE GenGridMode :
(
	none := 0,
	Grid := 1,
	GridDisconnected := 11,
	GridToNone := 12,
	Genset := 2
);
END_TYPE

// ---- POUs/MonitoringControl/ExternalControl/enums/uSWversion.TcDUT
TYPE uSWversion :
UNION
	a4byte_SWVer 	: 	ARRAY[0..3] OF BYTE;
	UD_SWVer		:	UDINT; 
END_UNION
END_TYPE

// ---- POUs/MonitoringControl/ExternalControl/Structs/future use/ST_PNInput_DCBusExpansion.TcDUT
TYPE ST_PNInput_DCBusExpansion :
STRUCT
	ControlBits	:	DWORD;
END_STRUCT
END_TYPE

// ---- POUs/MonitoringControl/ExternalControl/Structs/future use/ST_PNInput_DCCharger.TcDUT
TYPE ST_PNInput_DCCharger :
STRUCT
	Controlbits	:	DWORD;
	//b_enable?
	//b_resetCharger
	//b_StartCharging
	Powerlimit	:	DWORD;
END_STRUCT
END_TYPE

// ---- POUs/MonitoringControl/ExternalControl/Structs/future use/ST_PNInput_ParallelOperation.TcDUT
TYPE ST_PNInput_ParallelOperation :
STRUCT
	Controlbits			:	DWORD;
	//b_DetectSlaves	
	r_ActivePower		:	DWORD;
	r_reactivePower		:	DWORD;
END_STRUCT
END_TYPE

// ---- POUs/MonitoringControl/ExternalControl/Structs/future use/ST_PNOutput_DCCharger.TcDUT
TYPE ST_PNOutput_DCCharger :
STRUCT
	statusbits		:	DWORD;
	ChargerStatus	:	DWORD;
	ChargePower		:	DWORD;
END_STRUCT
END_TYPE

// ---- POUs/MonitoringControl/ExternalControl/Structs/future use/ST_PNOutput_DCExpansion.TcDUT
TYPE ST_PNOutput_DCExpansion :
STRUCT
	statusbits	: DWORD;
	Busvoltage	: DWORD;
	RatedPower	: DWORD;
	LoadPercentage	: DWORD;
	CurrentPower	: DWORD;
END_STRUCT
END_TYPE

// ---- POUs/MonitoringControl/ExternalControl/Structs/future use/ST_PNOutput_ParallelOperation.TcDUT
TYPE ST_PNOutput_ParallelOperation :
STRUCT
	statusbits		:	DWORD;
	ActivePower		:	DWORD;
	ReactivePower	:	DWORD;
END_STRUCT
END_TYPE

// ---- POUs/MonitoringControl/ExternalControl/Structs/NestedStructs/ST_PNInput_ACDCCharger.TcDUT
TYPE ST_PNInput_ACDCCharger :
STRUCT
	w_Control			:	WORD;
	ui_ACCurrentlimit	:	UINT	:=	0;
	UI_Pset				:	UINT	:=	0;
	ui_SocMaxLimit		:	UINT	:=	100;
	ui_MinGridVoltage	:	Uint	:=	360;
END_STRUCT
END_TYPE

// ---- POUs/MonitoringControl/ExternalControl/Structs/NestedStructs/ST_PNInput_Battery.TcDUT
TYPE ST_PNInput_Battery :
STRUCT
	w_Control		:	WORD;
	ui_SocMinLimit	:	UINT	:=	0;
	ui_SocMaxLimit	:	UINT	:=	100;
END_STRUCT
END_TYPE

// ---- POUs/MonitoringControl/ExternalControl/Structs/NestedStructs/ST_PNInput_GenControl.TcDUT
TYPE ST_PNInput_GenControl :
STRUCT
	w_Control			:	WORD;
	ui_SOCStart			:	UINT;
	ui_SOCStop			:	UINT;
	ui_BattLoadStart	:	UINT;
	ui_BattLoadStop		:	UINT;
	ui_GenPowerMode		:	UINT;
	ui_GenRatedPower	:	UINT;
	ui_GenMaxPowerLevel	:	UINT;
	ui_GenEffPowerLevel	:	UINT;
	ui_GenMinPowerLevel	:	UINT;
	ui_GenWarmupTime	:	UINT;
	ui_GenCooldownTime	:	UINT;
	ui_IsoPowerRamp		:	UINT;
	ui_GeneratorSetpoint : 	UINT;
	ui_StartStopControl	:	uint;	
END_STRUCT
END_TYPE

// ---- POUs/MonitoringControl/ExternalControl/Structs/NestedStructs/ST_PNInput_General.TcDUT
TYPE ST_PNInput_General :
STRUCT
	W_Control				:	WORD;
	ui_HeatBeat				:	UINT;
	ui_GridMode				:	UINT;
	ui_GridFormingSubMode	:	UINT;	
	ui_Earthingsystem		:	UINT;
	GridConnectionMode		:	UINT;
	PrimaryDigOutState		:	UINT := 99;
	SecondaryDigOutState	:	UINT := 99;
	PrimaryDigInState		:	UINT := 99;
	SecondaryDiginState		:	UINT := 99;
END_STRUCT
END_TYPE

// ---- POUs/MonitoringControl/ExternalControl/Structs/NestedStructs/ST_PNInput_InputField.TcDUT
TYPE ST_PNInput_InputField :
STRUCT
	w_Control				:	WORD;
	InputConnectionType		:	UINT;
//	ui_FeedInCurrentLimit	:	UINT;
//	ui_FeedOutCurrentLimit	:	UINT;
//	ui_IdleChargePower 		:	UINT;
//	ui_SocTarget			:	UINT;
//	ui_InputConnectionType	:	UINT;
END_STRUCT                       
END_TYPE

// ---- POUs/MonitoringControl/ExternalControl/Structs/NestedStructs/ST_PNInput_InputGridControl.TcDUT
TYPE ST_PNInput_InputGridControl :
STRUCT
	w_Control				:	WORD;
	ui_FeedInCurrentLimit	:	UINT;
	ui_SupplyCurrentLimit	:	UINT;
	ui_CurrentLimitRetries	:	UINT;
	ui_ContactorControl		:	uint;
END_STRUCT
END_TYPE

// ---- POUs/MonitoringControl/ExternalControl/Structs/NestedStructs/ST_PNInput_PeakShaveBox.TcDUT
TYPE ST_PNInput_PeakShaveBox :
STRUCT
	w_Control			:	WORD;
	ui_FeedInCurrentLimit	:	UINT;
	ui_SupplyCurrentLimit	:	UINT;
	ui_VTRatio				:	UINT;
	UI_CTRatio				:	UINT;
END_STRUCT
END_TYPE

// ---- POUs/MonitoringControl/ExternalControl/Structs/NestedStructs/ST_PNInput_Powerstack.TcDUT
TYPE ST_PNInput_Powerstack :
STRUCT
	w_Control			:	WORD;
	ui_NominalVoltage	:	UINT;
	ui_NominalFrequency	:	UINT;
	i_Pset				:	INT;
	i_Qset				:	INT;
	i_PFset				:	INT;
	ui_FrequencyDroop	:	UINT;
	ui_VoltageDroop		:	UINT;
	ui_PowerRampRate	:	UINT;
	ui_SOCDroopUpshiftStart		:	UINT;
	ui_SOCDroopDownShiftStart	:	UINT;
	ui_PowerLimitMode	:	UINT;
	ui_ACCurrentLimit	:	UINT;
END_STRUCT
END_TYPE

// ---- POUs/MonitoringControl/ExternalControl/Structs/NestedStructs/ST_PNOutput_ACDCCharger.TcDUT
TYPE ST_PNOutput_ACDCCharger :
STRUCT
	w_Status						: WORD;
	w_Warnings						: WORD;
	w_Faults						: WORD;
	ui_ChargerStatus				: WORD;
	TotalChargerPower				: WORD;
	AvailableChargePower			: UINT;
	ActivePower						: UINT;
	Frequency						: UINT;
	VoltageAB						: UINT;
	VoltageBC						: UINT;
	VoltageCA						: UINT;
	CurrentL1						: UINT;
	CurrentL2						: UINT;
	CurrentL3						: UINT;
	ui_ACCurrentLimitAct			: UINT;
	ui_PSetAct						: UINT;
	ui_SocLimitAct					: UINT;
	ui_MinGridVoltageAct			: UINT;
END_STRUCT
END_TYPE

// ---- POUs/MonitoringControl/ExternalControl/Structs/NestedStructs/ST_PNOutput_Battery.TcDUT
TYPE ST_PNOutput_Battery :
STRUCT
	ui_Status						: UINT;
	w_Warnings						: WORD;
	w_Faults						: WORD;

	ui_SOC							: UINT;
	ui_SOH							: UINT;
	ui_DClinkVoltage 				: UINT;
	i_DClinkCurrent 				: INT;
	ui_MaxAllowedDischargeCurrent 	: UINT;
	ui_MaxAllowedChargeCurrent 		: UINT;
	i_MinCellTemperature 			: INT;
	i_MaxCellTemperature			: INT;
	ui_RemainingChargeEnergy 		: UINT;
	ui_RemainingDischargeEnergy 	: UINT;
	ui_CycleCount					: UINT;
END_STRUCT
END_TYPE

// ---- POUs/MonitoringControl/ExternalControl/Structs/NestedStructs/ST_PNOutput_GenControl.TcDUT
TYPE ST_PNOutput_GenControl :
STRUCT
	w_Status					:	WORD;
	w_Warnings					:	WORD;
	w_Faults					:	WORD;
	ui_GeneratorStatus			:	UINT;	
END_STRUCT
END_TYPE

// ---- POUs/MonitoringControl/ExternalControl/Structs/NestedStructs/ST_PNOutput_General.TcDUT
TYPE ST_PNOutput_General :
STRUCT
	ui_SystemState				:	UINT;
	w_SystemStatus				:	WORD;	
	w_SystemWarnings			:	WORD;
	w_SystemFaults				:	WORD;
	w_CoolingSystemStatus		:	WORD;
	w_CoolingSystemWarnings		:	WORD;
	w_CoolingSystemFaults		:	WORD;
	w_InternalSupplyStatus		:	WORD;
	w_InternalSupplyWarnings	:	WORD;
	w_InternalSupplyFaults		:	WORD;	
	ui_HeartBeatOut				:	UINT;
	ui_Gridmode					: 	UINT;
	ui_GridFormingSubMode		: 	UINT;
	udi_SerialNumber			:	UDINT;
	dw_SWVersion				:	DWORD;
	//ui_InputConnectionType		:	UINT;
END_STRUCT
END_TYPE

// ---- POUs/MonitoringControl/ExternalControl/Structs/NestedStructs/ST_PNOutput_InputField.TcDUT
TYPE ST_PNOutput_InputField:
STRUCT
	w_Status					:	WORD;
	w_Warnings					:	WORD;
	w_Faults					:	WORD;
	ui_InputConnectionType		:	UINT;
	ui_InputConnectionState		:	UINT;
	i_ActivePower				:	INT;
	i_ReactivePower				:	INT;
	i_PowerFactor				:	INT;
	ui_Frequency				:	UINT;
	ui_VoltageL1N				:	UINT;
	ui_VoltageL2N				:	UINT;
	ui_VoltageL3N				:	UINT;
	ui_VoltageL1L2				:	UINT;
	ui_VoltageL2L3				:	UINT;
	ui_VoltageL3L1				:	UINT;
	ui_CurrentL1				:	UINT;
	ui_CurrentL2				:	UINT;
	ui_CurrentL3				:	UINT;
	ui_CurrentN					:	UINT;
	ui_CurrentLimitField		:	UINT;
	udi_TotalEnergySupplied 	:	UDINT;
	udi_TotalEnergyConsumed 	:	UDINT;
	ui_Current1L1				:	UINT;
	ui_Current1L2				:	UINT;
	ui_Current1L3				:	UINT;
	ui_Current1N				:	UINT;
	ui_Current2L1				:	UINT;
	ui_Current2L2				:	UINT;
	ui_Current2L3				:	UINT;
	ui_Current2N				:	UINT;
END_STRUCT
END_TYPE

// ---- POUs/MonitoringControl/ExternalControl/Structs/NestedStructs/ST_PNOutput_InputGridControl.TcDUT
TYPE ST_PNOutput_InputGridControl :
STRUCT
	w_Status					:	WORD;
	w_Warnings					:	WORD;
	w_Faults					:	WORD;
	ui_InputGridStatus			:	UINT;
END_STRUCT
END_TYPE

// ---- POUs/MonitoringControl/ExternalControl/Structs/NestedStructs/ST_PNOutput_OutputField.TcDUT
TYPE ST_PNOutput_OutputField:
STRUCT
	w_Status					:	WORD;
	w_Warnings					:	WORD;
	w_Faults					:	WORD;
	i_ActivePower				:	INT;
	i_ReactivePower				:	INT;
	i_PowerFactor				:	INT;
	ui_Frequency				:	UINT;
	ui_VoltageL1N				:	UINT;
	ui_VoltageL2N				:	UINT;
	ui_VoltageL3N				:	UINT;
	ui_VoltageL1L2				:	UINT;
	ui_VoltageL2L3				:	UINT;
	ui_VoltageL3L1				:	UINT;
	ui_CurrentL1				:	UINT;
	ui_CurrentL2				:	UINT;
	ui_CurrentL3				:	UINT;
	ui_CurrentN					:	UINT;
	ui_CurrentLimitField		:	UINT;
	udi_TotalEnergySupplied 	:	UDINT;
	udi_TotalEnergyConsumed 	:	UDINT;
	ui_Current1L1				:	UINT;
	ui_Current1L2				:	UINT;
	ui_Current1L3				:	UINT;
	ui_Current1N				:	UINT;
	ui_Current2L1				:	UINT;
	ui_Current2L2				:	UINT;
	ui_Current2L3				:	UINT;
	ui_Current2N				:	UINT;
	ui_Current3L1				:	UINT;
	ui_Current3L2				:	UINT;
	ui_Current3L3				:	UINT;
	ui_Current3N				:	UINT;
END_STRUCT
END_TYPE

// ---- POUs/MonitoringControl/ExternalControl/Structs/NestedStructs/ST_PNOutput_PeakShaveBox.TcDUT
TYPE ST_PNOutput_PeakShaveBox:
STRUCT
	w_Status					:	WORD;
	w_Warnings					:	WORD;
	w_Faults					:	WORD;
	i_ActivePower				:	INT;
	i_ReactivePower				:	INT;
	i_PowerFactor				:	INT;
	ui_Frequency				:	UINT;
	ui_VoltageL1N				:	UINT;
	ui_VoltageL2N				:	UINT;
	ui_VoltageL3N				:	UINT;
	ui_VoltageL1L2				:	UINT;
	ui_VoltageL2L3				:	UINT;
	ui_VoltageL3L1				:	UINT;
	ui_CurrentL1				:	UINT;
	ui_CurrentL2				:	UINT;
	ui_CurrentL3				:	UINT;
	ui_CurrentN					:	UINT;
END_STRUCT
END_TYPE

// ---- POUs/MonitoringControl/ExternalControl/Structs/NestedStructs/ST_PNOutput_PowerStack.TcDUT
TYPE ST_PNOutput_PowerStack :
STRUCT
	w_Status					:	WORD;
	w_Warnings					:	WORD;
	w_Faults					:	WORD;
	
	ui_PowerStackStatus			: UINT;
	i_ActivePower				: INT;
	i_ReactivePower				: INT;
	ui_SupplyVoltage			: UINT;
	ui_Supplyfrequency			: UINT;
	ui_ACCurrent				: UINT;
	i_PsetAct					: INT;
	i_QsetAct					: INT;
	i_PFSetAct					: UINT;
	ui_LoadPercentage			: UINT;
	ui_RatedCurrent				: UINT;
	ui_RatedPower				: UINT;
	ui_DischargePowerLimit		: UINT;
	ui_ChargePowerLimit			: UINT;
	ui_ACcurrentLimit			: UINT;
	ui_ApparentPowerLimit		: UINT;
	ui_ReactivePowerLimit		: UINT;
END_STRUCT
END_TYPE

// ---- POUs/MonitoringControl/ExternalControl/Structs/NestedStructs/ST_PNOutput_ZPT.TcDUT
TYPE ST_PNOutput_ZPT :
STRUCT
	w_Status					:	WORD;
	w_Warnings					:	WORD;
	w_Errors					:	WORD;
	ui_RatedPower				:	UINT;
	ui_Powerload				:	UINT;
	i_TransformerTemperature	:	INT;
END_STRUCT
END_TYPE

// ---- POUs/MonitoringControl/ExternalControl/Structs/ST_Extcontroller_params.TcDUT
TYPE ST_Extcontroller_params :
STRUCT
	b_BigEndian				: BOOL;
	b_testComm				: BOOL;
	b_MonitoringEnable		: BOOL := TRUE;
	b_ControlEnable			: BOOL := TRUE;
	w_CommTimeOut			: WORD := 10000; // milli seconds
	TestVars				: ST_PNTest;
	Limits					: ST_ExtController_limits;
END_STRUCT
END_TYPE

// ---- POUs/MonitoringControl/ExternalControl/Structs/ST_PNinput.TcDUT
TYPE ST_PNinput :
STRUCT
	PNIOBoxState		:	WORD;
	PNIOBoxDiag			:	WORD;	
	General 			: ST_PNInput_General;
	Battery				: ST_PNInput_Battery;
	Inputfield			: ST_PNInput_InputField;
	PSB					: ST_PNInput_PeakshaveBox;
	Powerstack			: ST_PNInput_Powerstack;
	GenControl 			: ST_PNInput_GenControl;
	InputGridControl	: ST_PNInput_InputGridControl;	
	ACDCCharger			: ST_PNInput_ACDCCharger;
END_STRUCT
END_TYPE

// ---- POUs/MonitoringControl/ExternalControl/Structs/ST_PNOutput.TcDUT
TYPE ST_PNOutput :
STRUCT
	General 		: ST_PNOutput_General;
	Battery			: ST_PNOutput_Battery;
	OutputField		: ST_PNOutput_Outputfield;
	InputField		: ST_PNOutput_Inputfield;
	Powerstack 		: ST_PNOutput_Powerstack;
	PSB 			: ST_PNOutput_PeakshaveBox;
	ZPT				: ST_PNOutput_ZPT;
	GenControl 		: ST_PNOutput_GenControl;
	InputGridControl: ST_PNOutput_InputGridControl;
	ACDCCharger		: ST_PNOutput_ACDCCharger;
END_STRUCT
END_TYPE

// ---- POUs/MonitoringControl/ExternalControl/Structs/ST_PNTest.TcDUT
TYPE ST_PNTest :
STRUCT
	b_CheckMonitoring	: BOOL;
	b_MonitoringOK		: BOOL;
	s_MonitoringErr		: STRING;
	i_Pset				: INT;
	i_Qset				: INT;
	w_SetAddress		: WORD;
	w_SetValue			: WORD;
	bit_start			: BOOL;
	bit_stop			: BOOL;
	bit_Shutdown		: BOOL;
	bit_SystemShutdown	: BOOL;
	bit_Reset			: BOOL;
	bit_EMStop			: BOOL;
	bit_AdvancedControl	: BOOL;
	bit_AutoSwitching	: BOOL;
	bit_Transportmode	: BOOL;
END_STRUCT
END_TYPE

// ---- POUs/MonitoringControl/HMI/_Structs/ControlStructures/OperationVars/ST_OperationVars.TcDUT
TYPE ST_OperationVars :
STRUCT
		inputgrid				: ST_OperationVars_Grid;
		Genset					: ST_OperationVars_Genset;
		PSB						: ST_OperationVars_Grid;
		charger					: ST_OperationVars_DCcharger;
		system					: ST_OperationVars_System;
		parallel				: ST_OperationVars_ParallelOperation;	
		BMS						: ST_OperationVars_BMS;	
END_STRUCT
END_TYPE

// ---- POUs/MonitoringControl/HMI/_Structs/ControlStructures/OperationVars/ST_OperationVars_BMS.TcDUT
TYPE ST_OperationVars_BMS :
STRUCT
	b_ManualStartHVDC	: BOOL;
END_STRUCT
END_TYPE

// ---- POUs/MonitoringControl/HMI/_Structs/ControlStructures/OperationVars/ST_OperationVars_DCcharger.TcDUT
TYPE ST_OperationVars_DCcharger :
STRUCT
	b_StartCharging						: BOOL;
	b_ResetCharger						: BOOL;
END_STRUCT
END_TYPE

// ---- POUs/MonitoringControl/HMI/_Structs/ControlStructures/OperationVars/ST_OperationVars_Genset.TcDUT
TYPE ST_OperationVars_Genset :
STRUCT 
	b_manualStart			: BOOL;
END_STRUCT
END_TYPE

// ---- POUs/MonitoringControl/HMI/_Structs/ControlStructures/OperationVars/ST_OperationVars_Grid.TcDUT
TYPE ST_OperationVars_Grid:
STRUCT
	b_SyncClose							: BOOL;
END_STRUCT
END_TYPE

// ---- POUs/MonitoringControl/HMI/_Structs/ControlStructures/OperationVars/ST_OperationVars_ParallelOperation.TcDUT
TYPE ST_OperationVars_ParallelOperation :
STRUCT
	b_DetectSlaves					: BOOL;
	
	
	// VDL ONLY
	r_ActivePowerSlave1				: REAL;
	r_ReactivePowerSlave1			: REAL;
	r_ActivePowerSlave2				: REAL;
	r_ReactivePowerSlave2			: REAL;
END_STRUCT
END_TYPE

// ---- POUs/MonitoringControl/HMI/_Structs/ControlStructures/OperationVars/ST_OperationVars_System.TcDUT
TYPE ST_OperationVars_System :
STRUCT
	//Powerstack
	r_NominalVoltage				: REAL := Settings.GridParams.r_GridNominalVoltage; //VAC
	r_NominalFrequency				: REAL := Settings.GridParams.r_GridNominalFrequency; //Hz
	
	//Power setpoints
	r_Pset							: REAL;// active power setpoint
	r_Qset							: REAL;// reactive power setpoint
	r_PFset							: REAL := 1;// powerfactor -1 .. 1
	b_PFsetEnable					: BOOL := TRUE;
	
	b_SounderMute					: BOOL;
	b_SounderTest					: BOOL;	
	
	//Mode transition
	b_GenGridModeTrans				: BOOL;	
	b_GridTakeOverEnable			: BOOL;
END_STRUCT
END_TYPE

// ---- POUs/MonitoringControl/HMI/_Structs/ControlStructures/ST_ControlsHMIonly.TcDUT
TYPE ST_ControlsHMIonly:
STRUCT
	b_Pup							: BOOL;
	b_Pdown							: BOOL;
	b_Qup							: BOOL;
	b_Qdown							: BOOL;
	b_QReset						: BOOL;
	b_PReset						: BOOL;
	b_HMITaskKill					: BOOL;
	b_ActivateSetting				: BOOL;
END_STRUCT
END_TYPE

// ---- POUs/MonitoringControl/HMI/_Structs/ControlStructures/ST_ControlVars.TcDUT
TYPE ST_ControlVars :
STRUCT
	b_start							: BOOL;
	b_stop							: BOOL;
	b_shutdown						: BOOL;
	b_Reset							: BOOL;
	b_SystemShutdown				: BOOL;
	b_EMstop						: BOOL;
	b_ClearHistory					: BOOL;
	b_ActivateSettings 				: BOOL;
	b_ActivateIotSettings			: BOOL;
	b_startDeHum					: BOOL;
END_STRUCT
END_TYPE

// ---- POUs/MonitoringControl/HMI/_Structs/MonitoringStructures/ST_HMIdata.TcDUT
TYPE ST_HMIdata :
STRUCT
	s_Type		: STRING(12);
	s_Name		: STRING(25);
	s_Data		: STRING(12);
	s_Unit		: STRING(4);
	b_Warning	: BOOL; 
END_STRUCT
END_TYPE

// ---- POUs/MonitoringControl/HMI/_Structs/MonitoringStructures/ST_HMI_ConditionalFormatting.TcDUT
TYPE ST_HMI_ConditionalFormatting :
STRUCT
	b_ShowPset			: BOOL;
	b_ShowQset			: BOOL;
	b_showPFset			: BOOL;
	b_ShowInputDisconnect: BOOL;
	b_ShowGenManStartStop: BOOL;
	b_ShowShowGensetInfo : BOOL;
	b_EnableTNCheckBox 		: BOOL;
	b_ShowExtgenset		: BOOL;
	b_TransportModeActive : BOOL;
	b_ShowGensetHybridMode: BOOL;
	b_showPSBData			: BOOL;
	b_showModetransbutton	: BOOL;
END_STRUCT
END_TYPE

// ---- POUs/MonitoringControl/HMI/_Structs/MonitoringStructures/ST_HMI_Monitor_AcDcCharger.TcDUT
TYPE ST_HMI_Monitor_AcDcCharger :
STRUCT
	state 			: STRING;
	available 		: BOOL;
	r_AcCurrentMax	: REAL;
	r_AcPowerMax	: REAL;
	r_DcPower 		: REAL;
	r_AcPower 		: REAL;
	r_AcCurrent		: REAL;
	r_AcVoltage		: REAL;
END_STRUCT
END_TYPE

// ---- POUs/MonitoringControl/HMI/_Structs/MonitoringStructures/ST_HMI_Monitor_Arraydata.TcDUT
TYPE ST_HMI_Monitor_Arraydata :
STRUCT
	ACInputData			: ARRAY [1..35] OF ST_HMIData;
	ACOutputData		: ARRAY [1..36] OF ST_HMIData;
	AcDcChargerData		: ARRAY [1..13] OF ST_HMIData;
	DcExtension			: ARRAY [1..4] OF ST_HMIData;
	PowerstackData 		: ARRAY [1..20] OF ST_HMIData;
	PmMasterData		: ARRAY [1..58] OF ST_HMIData;
	PmSlaveData			: ARRAY [1..58] OF ST_HMIData;
	PNcontrolData		: ARRAY [1..45] OF ST_HMIData;
	IotcontrolData		: ARRAY [1..45] OF ST_HMIData;
	PSBdata				: ARRAY [1..24] OF ST_HMIData;
	MBMUdata			: ARRAY [1..20] OF ST_HMIData;
	SBMU1Data			: ARRAY [1..21] OF ST_HMIData;
	SBMU2Data			: ARRAY [1..21] OF ST_HMIData;
	SBMU3Data			: ARRAY [1..21] OF ST_HMIData;
	SBMU4Data			: ARRAY [1..21] OF ST_HMIData;
	CoolingSystem		: ARRAY [1..5] OF ST_HMIData;
	CoolingSystemHp1	: ARRAY [1..10] OF ST_HMIData;
	CoolingSystemHp2	: ARRAY [1..10] OF ST_HMIData;
	Genset				: ARRAY [1..14] OF ST_HMIData;
END_STRUCT
END_TYPE

// ---- POUs/MonitoringControl/HMI/_Structs/MonitoringStructures/ST_HMI_Monitor_ArrayDataFormat.TcDUT
TYPE ST_HMI_Monitor_ArrayDataFormat :
STRUCT
	s_name				: STRING(25);
	s_type				: STRING(12);
	s_unit				: STRING(12);
	r_data				: REAL;
	i_precision			: INT := -1;
	b_warning			: BOOL;
END_STRUCT
END_TYPE

// ---- POUs/MonitoringControl/HMI/_Structs/MonitoringStructures/ST_HMI_Monitor_Battery.TcDUT
TYPE ST_HMI_Monitor_Battery :
STRUCT
	e_status			: eBMS_Status;
	r_SocScaled			: REAL := 10; 
	r_SoCReal			: REAL;
	r_CellVoltageMax	: REAL;
	r_CellVoltageMin	: REAL;
	r_CellTempMax		: REAL;
	r_CellTempMin		: REAL;
	r_MaxDischargePower	: REAL;
	r_MaxChargePower	: REAL;
	r_DCvoltage			: REAL;
	r_DCcurrent			: REAL;
	r_SoH				: REAL;
	r_NetRemainingCapacity: REAL; //kWh
	ui_CycleCount		: UINT;
	
END_STRUCT
END_TYPE

// ---- POUs/MonitoringControl/HMI/_Structs/MonitoringStructures/ST_HMI_Monitor_Connections.TcDUT
TYPE ST_HMI_Monitor_Connections :
STRUCT
	b_ExtControllerEnabled		: BOOL;
	e_ExtConnectionState		: eConnectionState;
	s_OutputJson				: STRING(2000);
	b_IoTEnabled				: BOOL;
	e_IoTConnectionState		: eConnectionState;
	b_PsbOK						: BOOL;			
	e_ActiveController			: eControlSources;
	e_ProfinetState				: eNetcomState;
	e_EthercatState				: eNetcomState;
	r_CPUload					: REAL;
	
END_STRUCT
END_TYPE

// ---- POUs/MonitoringControl/HMI/_Structs/MonitoringStructures/ST_HMI_Monitor_CoolingSystem.TcDUT
TYPE ST_HMI_Monitor_CoolingSystem :
STRUCT
	e_OperationMode 		: eCoolingSystemState;
	e_HeatPumpStatus		: eHeatPumpState;
	r_CoolantTemperature	:	REAL;
	r_CoolantPressure		:	REAL;
	r_EnclosureDewpoint		:	REAL;
	b_HeatPumpError			: 	BOOL;
	b_HeatPumpWarning		:	BOOL;
	b_CoolantPressureWarning: 	BOOL;
	b_CoolantPressureError	:	BOOL;
	b_CoolantTempWarning	: 	BOOL;
END_STRUCT
END_TYPE

// ---- POUs/MonitoringControl/HMI/_Structs/MonitoringStructures/ST_HMI_Monitor_DcLink.TcDUT
TYPE ST_HMI_Monitor_DcLink :
STRUCT
	state 			: STRING;
	available 		: BOOL;
	//r_AcCurrentMax	: REAL;
	//r_AcPowerMax	: REAL;
	//r_DcPower 		: REAL;
	//r_AcPower 		: REAL;
	//r_AcCurrent		: REAL;
	//r_AcVoltage		: REAL;
	
	r_CurrentShunt		: REAL;
	r_TempratureShunt	: REAL;
	r_PowerShunt		: REAL;
	r_ChargeShunt		: REAL;
	r_BusVoltageShunt	: REAL;
	r_EnergyShunt		: REAL;  
END_STRUCT
END_TYPE

// ---- POUs/MonitoringControl/HMI/_Structs/MonitoringStructures/ST_HMI_Monitor_Enclosure.TcDUT
TYPE ST_HMI_Monitor_Enclosure :
STRUCT
	//Doors
	b_DoorClosedClientPanel		: BOOL;
	b_DoorClosedControlPanel	: BOOL;
	b_DoorClosedInverter		: BOOL;
	
	//climate
	r_Humidity					: REAL := -255;
	r_Temperature				: REAL := -255;
	b_HumidityHigh				: BOOL;
	b_HumidityTooHigh			: BOOL;
	b_TemperatureHigh			: BOOL;
	b_TemperatureTooHigh		: BOOL;
	b_TemperatureLow			: BOOL;
	b_TemperatureTooLow			: BOOL;
	
END_STRUCT
END_TYPE

// ---- POUs/MonitoringControl/HMI/_Structs/MonitoringStructures/ST_HMI_Monitor_FireDetection.TcDUT
TYPE ST_HMI_Monitor_FireDetection :
STRUCT
	e_SmokeDetectorState			: eSmokeDetectAlarmStatus;
	e_CoDetectorState				: eCOAlarmStatus;
	r_CoDetectorLeftValue			: REAL; //ppm
	r_CoDetectorRightValue			: REAL; //ppm			
END_STRUCT
END_TYPE

// ---- POUs/MonitoringControl/HMI/_Structs/MonitoringStructures/ST_HMI_Monitor_IPSU.TcDUT
TYPE ST_HMI_Monitor_IPSU :
STRUCT
	b_24VdcOK			: BOOL;
	b_400VacOK			: BOOL;
	b_HvdcOK			: BOOL;
	b_GridFuseOK		: BOOL;
	b_CeeFuseOK			: BOOL;
	e_400VSource		: e400VSupplySource;
END_STRUCT
END_TYPE

// ---- POUs/MonitoringControl/HMI/_Structs/MonitoringStructures/ST_HMI_Monitor_Limits.TcDUT
TYPE ST_HMI_Monitor_Limits :
STRUCT
	//LIMITS
	//r_Pmin						: REAL ;
	//r_Pmax						: REAL ;
	//r_QMin						: REAL ;
	//r_QMax						: REAL ;
	r_ACcurrentLimit			: REAL;
	r_ApparentPowerlimit		: REAL;
	r_ActivePowerlimit			: REAL;
	r_DCcurrentLimit			: REAL;
	r_DroopLimit				: REAL;
	
END_STRUCT
END_TYPE

// ---- POUs/MonitoringControl/HMI/_Structs/MonitoringStructures/ST_HMI_Monitor_OCP.TcDUT
TYPE ST_HMI_Monitor_OCP : //overcurrent protection
STRUCT
	b_InputMCCBstate			: BOOL;
	b_OutputMCCBstate			: BOOL;
	b_InputOverloadWarning		: BOOL;
	b_InputOverloadAlarm		: BOOL;
	b_OutputOverloadWarning		: BOOL;
	b_OutputOverloadAlarm		: BOOL;
	s_Location					: STRING;
	r_CurrentPeak				: REAL;
	t_PeakDuration				: TIME;	
END_STRUCT
END_TYPE

// ---- POUs/MonitoringControl/HMI/_Structs/MonitoringStructures/ST_HMI_Monitor_Powerstack.TcDUT
TYPE ST_HMI_Monitor_Powerstack :
STRUCT
	// stack
	r_Powerload					: REAL;
	r_DcPower					: REAL;
	r_ActivePower				: REAL;
	r_throttlingValue			: REAL;
	
	b_ACDetected				: BOOL;
	b_DCDetected				: BOOL;
	b_StartedState				: BOOL;
	b_islandOperation			: BOOL;
	b_ControlEnabled			: BOOL;
	e_NetContState				: eNetContactorState;
	e_ACrotationState			: eACRotationState;
	e_StatusPowerStack			: eStatusPowerstack;
	
	//Master
	b_MasterEnabled				: BOOL;
	b_MasterWarning				: BOOL;
	b_MasterMCCBfb				: BOOL;
	e_MasterState				: eStatusPowerModule;
	r_MasterthrotValue			: REAL;
	b_MasterTempThrotActive		: BOOL;
	b_MasterCurrThrotActive		: BOOL;		
	
	
	b_SlaveEnabled				: BOOL;
	b_SlaveWarning				: BOOL;
	b_SlaveMCCBfb				: BOOL;
	e_SlaveState				: eStatusPowerModule;
	r_SlavethrotValue			: REAL;
	b_SlaveTempThrotActive		: BOOL;
	b_SlaveCurrThrotActive		: BOOL;		
	
END_STRUCT
END_TYPE

// ---- POUs/MonitoringControl/HMI/_Structs/MonitoringStructures/ST_HMI_Monitor_Protections.TcDUT
TYPE ST_HMI_Monitor_Protections :
STRUCT
	b_MrcdbOK					: BOOL;
	b_MrcdbWarning				: BOOL;
	b_MrcdbAlarm				: BOOL;
	b_InsulationEnable			: BOOL;
	b_InsulationOk				: BOOL;
	b_InsulationWarning			: BOOL;
	b_InsulationAlarm			: BOOL;
	b_InsulationPenDetected		: BOOL; //discrepence of PEN config and detected situation
	e_EarthingSystemDetected	: eEarthingSystems; //0: Unknown, 1: TN-S, 2: TN-C, 3: IT.
	b_SurgeType12OK				: BOOL;
	b_SurgeType3OK				: BOOL;
END_STRUCT
END_TYPE

// ---- POUs/MonitoringControl/HMI/_Structs/MonitoringStructures/ST_HMI_Monitor_PSB.TcDUT
TYPE ST_HMI_Monitor_PSB :
STRUCT
	b_Connected : BOOL;
	b_Active	: BOOL;
END_STRUCT
END_TYPE

// ---- POUs/MonitoringControl/HMI/_Structs/MonitoringStructures/ST_HMI_Monitor_switchgear.TcDUT
TYPE ST_HMI_Monitor_switchgear :
STRUCT
	//Switchgear
	b_ACDetectedBusbar			: BOOL;
	b_ACDetectedInput			: BOOL;
	b_DCDetected				: BOOL;
	b_PeNeutralLink				: BOOL;
	b_ACInputState				: BOOL; //summary of MCCB and contactor state.
	b_InputSync					: BOOL;
	r_ACInputPower				: REAL;
	b_NetContactorState			: BOOL; //summary of netcontactor left and right close state.
	b_ACOutputState				: BOOL;
	r_ACOutputPower				: REAL; 
	b_DCCouplingState			: BOOL;
	r_DCCouplingCurrent			: REAL;
END_STRUCT
END_TYPE

// ---- POUs/MonitoringControl/HMI/_Structs/MonitoringStructures/ST_HMI_Monitor_System.TcDUT
TYPE ST_HMI_Monitor_System :
STRUCT
	r_currentEfficiency		: REAL;
	r_averageEfficiency		: REAL;
	r_RountripEfficiency	: REAL;
	r_DischargeEnergy		: REAL;
	r_ChargedEnergy			: REAL;
	
	e_SystemState			: eSystemState; //0:Idle, 1: Stand-by, 2:Conditioning, 3:Dry-Cycle, 4: Running, 5: Charging only, 6: Discharging only, 7: Stopped 8:Fault
	e_GridMode				: eGridmode;
	e_UgridPowermode		: eUgridPowermode;
	
	b_EarthingSelected		: BOOL;
	b_startAllowed			: BOOL;
	
	b_Alert					: BOOL;
	b_SMSnumberConfigured	: BOOL;
	b_CustomNameConfigured	: BOOL;
	b_TransportModePending	: BOOL;
	b_MasterSlaveModeEnabled: BOOL;
	
	s_SystemName			: STRING(20);
END_STRUCT
END_TYPE

// ---- POUs/MonitoringControl/HMI/_Structs/MonitoringStructures/ST_HMI_Monitor_UPS.TcDUT
TYPE ST_HMI_Monitor_UPS :
STRUCT
	b_ChargerActive		: BOOL;
	b_SupplyOnBattery	: BOOL;
	r_InputVoltage		: REAL;
	r_OutputVoltage		: REAL;
	r_OutputCurrent		: REAL;
	r_BatteryVoltage	: REAL;
	b_InputVoltageFault	: BOOL;
	b_BatteryLowInfo	: BOOL;
	b_BatteryLowWarning : BOOL;
	b_BatteryLowCritical: BOOL;
	ui_SoC				: UINT;
END_STRUCT
END_TYPE

// ---- POUs/MonitoringControl/HMI/_Structs/MonitoringStructures/ST_HMI_Monitor_ZPT.TcDUT
TYPE ST_HMI_Monitor_ZPT :
STRUCT
	b_ZPTOverloadWarning	: BOOL;
	b_ZPTOverloadAlarm		: BOOL;
	b_VoltageUnbalanceWarning: BOOL;
	b_VoltageUnbalanceAlarm	: BOOL;
	r_TemperatureL1			: REAL;
	b_TempWarningL1			: BOOL;
	b_TempAlarmL1			: BOOL;
	r_TemperatureL2			: REAL;
	b_TempWarningL2			: BOOL;
	b_TempAlarmL2			: BOOL;
	r_TemperatureL3			: REAL;
	b_TempWarningL3			: BOOL;
	b_TempAlarmL3			: BOOL;
	r_powerload				: REAL;	//%
	r_voltageunbalance		: REAL; //%
END_STRUCT
END_TYPE

// ---- POUs/MonitoringControl/HMI/_Structs/MonitoringStructures/ST_HMI_PowerMeas.TcDUT
TYPE ST_HMI_PowerMeas :
STRUCT
	Voltage			: REAL;
	Frequency		: REAL;
	ActivePower		: REAL;
	ReactivePower	: REAL;
	Current			: REAL;
END_STRUCT
END_TYPE

// ---- POUs/MonitoringControl/HMI/_Structs/MonitoringStructures/ST_HMI_PowerMeasDC.TcDUT
TYPE ST_HMI_PowerMeasDC :
STRUCT
	Voltage : REAL;
	Current	: REAL;
	Power	: REAL;
	SOC		: REAL;
END_STRUCT
END_TYPE

// ---- POUs/MonitoringControl/HMI/_Structs/ST_HMI_Control.TcDUT
TYPE ST_HMI_Control EXTENDS ST_System_Control:
STRUCT
	HMIonly				: ST_ControlsHMIonly;
END_STRUCT
END_TYPE

// ---- POUs/MonitoringControl/HMI/_Structs/ST_HMI_Historize.TcDUT
TYPE ST_HMI_Historize :
STRUCT
	PSB				: ST_HMI_PowerMeas;
	Input			: ST_HMI_PowerMeas;
	Output			: ST_HMI_PowerMeas;
	Inverter		: ST_HMI_PowerMeas;
	Battery			: ST_HMI_PowerMeasDC;
	Charger			: ST_HMI_PowerMeas;
	DcCoupling		: ST_HMI_PowerMeasDC;
END_STRUCT
END_TYPE

// ---- POUs/MonitoringControl/HMI/_Structs/ST_HMI_Monitor.TcDUT
//CHANGING THESE VARIABLES WILL RESULT IN BROKEN LINKS TO THE HMI!
TYPE ST_HMI_Monitor :
STRUCT
	ConditionalFormatting		: ST_HMI_ConditionalFormatting;
	System						: ST_HMI_Monitor_System;
	Powerstack					: ST_HMI_Monitor_Powerstack;
	enclosure					: ST_HMI_Monitor_enclosure;
	firedetection				: ST_HMI_Monitor_Firedetection;
	IPSU						: ST_HMI_Monitor_IPSU;
	OCP							: ST_HMI_Monitor_OCP;
	UPS							: ST_HMI_Monitor_UPS;
	protections					: ST_HMI_Monitor_protections;
	ZPT							: ST_HMI_Monitor_ZPT;
	Switchgear					: ST_HMI_Monitor_switchgear;
	Battery						: ST_HMI_Monitor_Battery;					
	Limits						: ST_HMI_Monitor_limits;
	Connections					: ST_HMI_Monitor_Connections;
	arraydata					: ST_HMI_Monitor_Arraydata;
	cooling						: ST_HMI_Monitor_CoolingSystem;
	AcDcCharger					: ST_HMI_Monitor_AcDcCharger;
	Powercontroller				: ST_PowerControl_Get;
	GenGridController			: ST_GenGridController_get;
	controlfb					: ST_ControlVars;
	PSB							: ST_HMI_Monitor_PSB;	
	DcLink 						: ST_HMI_Monitor_DcLink;
	b_testBool					: BOOL;
END_STRUCT
END_TYPE

// ---- POUs/MonitoringControl/IoT/DUTS/eConnectionState.TcDUT
{attribute 'qualified_only'}
{attribute 'strict'}
{attribute 'to_string'}
 
TYPE eConnectionState :
(
	disconnected := 0,			// no mqtt connection established
	connected	:= 1,			 // connected but not authorized yet
	authorization_declined := 2, // connected but authorization failed
	authorized	:= 3			// connected and authorized
);
END_TYPE

// ---- POUs/MonitoringControl/IoT/DUTS/eDataMappingVarNames.TcDUT
{attribute 'qualified_only'}
{attribute 'to_string'}

TYPE eDataMappingVarNames :
(*
 * Enumeration for mapping every variable in ST_System_Monitor to a fixed
 * monitoring ID.  The hierarchy is fully expanded at every nesting level.
 *
 * Naming convention:
 *   Structs : <topLevel>_<field>_<subField>_..._<leafField>
 *   Arrays  : <path>_<indexName>  where the index names are:
 *               _AVG      (index 0)
 *               _L1       (index 1)
 *               _L2       (index 2)
 *               _L3       (index 3)
 *               _N        (index 4)
 *               _minimum  (index 5)
 *               _maximum  (index 6)
 *   Only electrical measurement arrays are individually expanded:
 *   ar_ActivePower, ar_ReactivePower, ar_ApparentPower,
 *   ar_PhaseVoltage, ar_LineVoltage, ar_Current,
 *   ar_Frequency, ar_THD, ar_PowerFactor.
 *   The aggregate array variable is NOT included; only individual
 *   per-index entries are present (e.g. ar_Current_AVG, ar_Current_L1).
 *
 *)
(	
None													:= 0,
	(*═════════════════════════════════════════════════════════*)
	(*  Safety and System State    *)
	(*═════════════════════════════════════════════════════════*)
	safety_b_SafetyOK                                          , (* BOOL *)
	safety_b_EstopChannelAOK                                   , (* BOOL *)
	safety_b_EstopChannelBOK                                   , (* BOOL *)
	safety_b_InsulationMonitorOK                               , (* BOOL *)
	safety_b_MRCDBOK                                           , (* BOOL *)
	safety_b_InverterDoorOK                                    , (* BOOL *)
	safety_b_ZptOK                                             , (* BOOL *)
	system_b_SMSnumberConfigured                               , (* BOOL *)
	system_b_CustomNameConfigured                              , (* BOOL *)
	system_s_SystemName                                        , (* STRING(20) *)
	system_b_TransportModePending                              , (* BOOL *)
	system_b_DehumModePending                                  , (* BOOL *)
	system_e_State                                             , (* eSystemState *)
	system_e_gridmode                                          , (* eGridmode *)
	system_e_UgridPowermode                                    , (* eUgridPowermode *)
	system_b_StartAllowed                                      , (* BOOL *)
	system_r_CurrentEfficiency                                 , (* REAL *)
	system_r_AvgEfficiency                                     , (* REAL *)
	system_r_RoundtripEfficiency                               , (* REAL *)
	system_DT_SystemTime                                       , (* DT *)
	system_PowerController_r_CurrentAct                        , (* REAL *)
	system_PowerController_r_Sact                              , (* REAL *)
	system_PowerController_r_PAct                              , (* REAL *)
	system_PowerController_r_QAct                              , (* REAL *)
	system_PowerController_r_PhaseVoltageAct                   , (* REAL *)
	system_PowerController_r_PFact                             , (* REAL *)
	system_PowerController_r_FeedInCurrentLimitActual          , (* REAL *)
	system_PowerController_r_SupplyInCurrentLimitActual        , (* REAL *)
	system_PowerController_b_ThrottlingActive                  , (* BOOL *)
	system_PowerController_ui_ThrottlingType                   , (* UINT *)
	system_PowerController_events_b_ReactivePIDError           , (* BOOL *)
	system_PowerController_events_b_ActivePIDError             , (* BOOL *)
	system_PowerController_events_b_FreqShiftPIDError          , (* BOOL *)
	system_GenGridController_b_active                          , (* BOOL *)
	system_GenGridController_b_faultActive                     , (* BOOL *)
	system_GenGridController_b_gensetHot                       , (* BOOL *)
	system_GenGridController_b_gensetStarting                  , (* BOOL *)
	system_GenGridController_b_ModeTransActive                 , (* BOOL *)
	system_GenGridController_b_ModeTransInhibit                , (* BOOL *)
	system_GenGridController_b_ModeChanged                     , (* BOOL *)
	system_GenGridController_b_ShowModeTrans                   , (* BOOL *)
	system_GenGridController_b_extGensetMode                   , (* BOOL *)
	system_GenGridController_b_gensetcontrol                   , (* BOOL *)
	system_GenGridController_e_BreakerMode                     , (* eBreakerOperationMode *)
	system_GenGridController_e_PowerControlMode                , (* ePowerControlMode *)
	system_GenGridController_e_GensetMode                      , (* eGensetMode *)
	system_GenGridController_e_GensetStartStop                 , (* eGensetStartStop *)
	system_GenGridController_e_state                           , (* eGenGridState *)
	system_GenGridController_e_RunCondition                    , (* eRunCondition *)
	system_GenGridController_events_b_InvalidGensetParameters  , (* BOOL *)
	system_GenGridController_events_b_RotationFieldFault       , (* BOOL *)
	system_GenGridController_events_b_CurrentLimitDisconnect   , (* BOOL *)
	system_GenGridController_events_b_CurrentLimitTrip         , (* BOOL *)
	system_GenGridController_events_b_EmstopDisconnect         , (* BOOL *)
	system_GenGridController_events_b_ShutdownDisconnect       , (* BOOL *)
	system_GenGridController_events_b_OverloadTrip             , (* BOOL *)
	system_GenGridController_events_b_OverFreqTrip             , (* BOOL *)
	system_GenGridController_events_b_UnderFreqTrip            , (* BOOL *)
	system_GenGridController_events_b_OverVoltTrip             , (* BOOL *)
	system_GenGridController_events_b_UnderVoltTrip            , (* BOOL *)
	system_GenGridController_events_b_ShutdownTimeOut          , (* BOOL *)
	system_GenGridController_events_b_SynchronisationFault     , (* BOOL *)
	system_GenGridController_events_b_StartupFault             , (* BOOL *)
	system_GenGridController_events_b_WarmupFault              , (* BOOL *)
	system_GenGridController_events_b_GenDownTrip              , (* BOOL *)
	system_GenGridController_events_b_GridLostTrip             , (* BOOL *)
	system_GenGridController_events_b_TransToGenIsoInhibit     , (* BOOL *)
	system_GenGridController_events_b_TransToGenDroopInhibit   , (* BOOL *)
	system_GenGridController_events_b_TransToGenFixInhibit     , (* BOOL *)
	system_GenGridController_events_b_TransFromInputGridAckRQ  , (* BOOL *)
	system_GenGridController_events_b_TransFromInputGenAckRQ   , (* BOOL *)
	system_GenGridController_events_b_StartingInhibit          , (* BOOL *)
	system_events_b_RestartRequiredMachineName                 , (* BOOL *)
	system_events_b_TimeUpdateFailed                           , (* BOOL *)

